PROGRAM MAIN
VAR
END_VAR

END_PROGRAM

(* stored: Version 1.1.0.1, ProductVersion 3.1.0.38
   POU MAIN: Id {77f10f75-832a-434f-942b-0770252a3379}, SpecialFunc None *)
